// LS Electric XG5000 project: project
// PLC LSPLC

PROGRAM NewProgram (task: 스캔 프로그램)

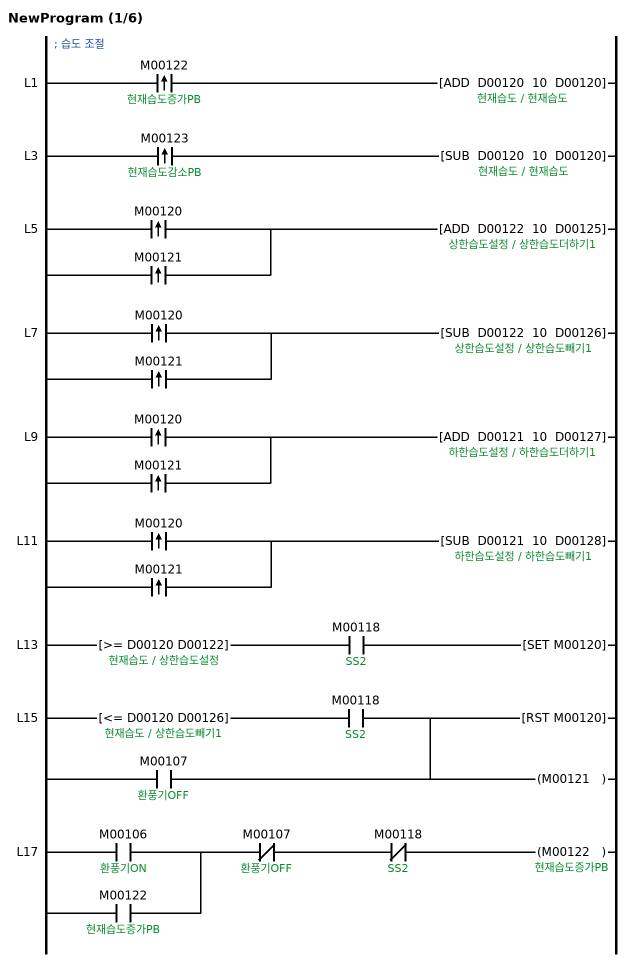
// 습도 조절
; L1
LOADP     M00122	// 현재습도증가PB
ADD       D00120 10 D00120	// 현재습도 / 현재습도
; L3
LOADP     M00123	// 현재습도감소PB
SUB       D00120 10 D00120	// 현재습도 / 현재습도
; L5
LOADP     M00120
ORP       M00121
ADD       D00122 10 D00125	// 상한습도설정 / 상한습도더하기1
; L7
LOADP     M00120
ORP       M00121
SUB       D00122 10 D00126	// 상한습도설정 / 상한습도빼기1
; L9
LOADP     M00120
ORP       M00121
ADD       D00121 10 D00127	// 하한습도설정 / 하한습도더하기1
; L11
LOADP     M00120
ORP       M00121
SUB       D00121 10 D00128	// 하한습도설정 / 하한습도빼기1
; L13
LOAD>=    D00120 D00122	// 현재습도 / 상한습도설정
AND       M00118	// SS2
SET       M00120
; L15
LOAD<=    D00120 D00126	// 현재습도 / 상한습도빼기1
AND       M00118	// SS2
OR        M00107	// 환풍기OFF
RST       M00120
OUT       M00121
; L17
LOAD      M00106	// 환풍기ON
OR        M00122	// 현재습도증가PB
AND NOT   M00107	// 환풍기OFF
AND NOT   M00118	// SS2
OUT       M00122	// 현재습도증가PB

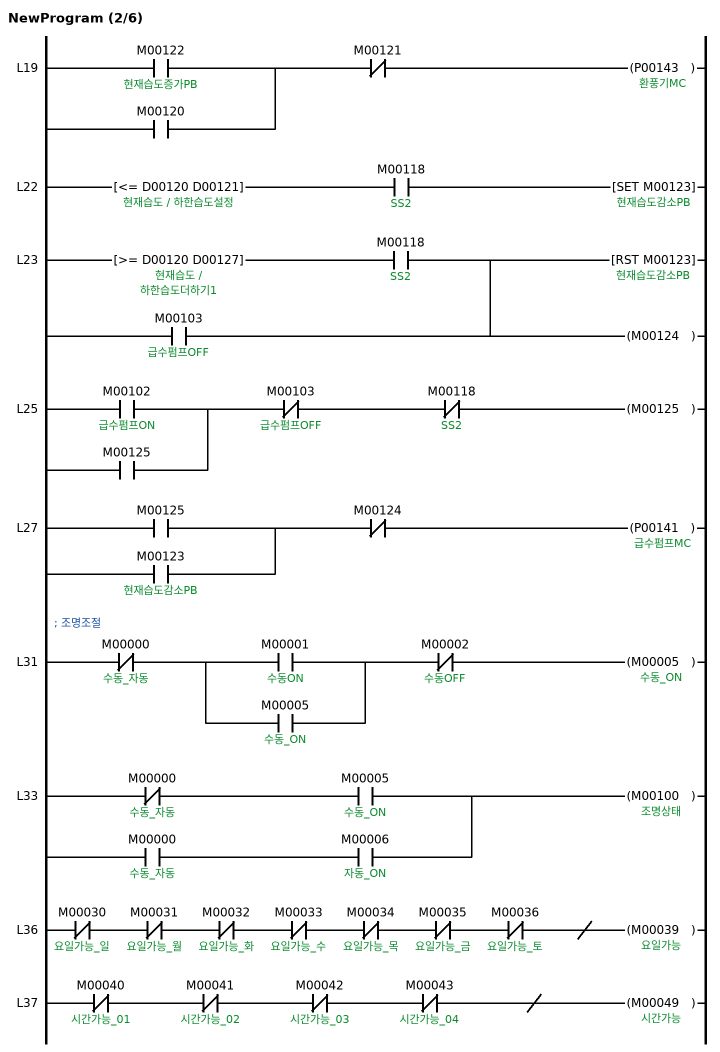
; L19
LOAD      M00122	// 현재습도증가PB
OR        M00120
AND NOT   M00121
OUT       P00143	// 환풍기MC
; L22
LOAD<=    D00120 D00121	// 현재습도 / 하한습도설정
AND       M00118	// SS2
SET       M00123	// 현재습도감소PB
; L23
LOAD>=    D00120 D00127	// 현재습도 / 하한습도더하기1
AND       M00118	// SS2
OR        M00103	// 급수펌프OFF
RST       M00123	// 현재습도감소PB
OUT       M00124
; L25
LOAD      M00102	// 급수펌프ON
OR        M00125
AND NOT   M00103	// 급수펌프OFF
AND NOT   M00118	// SS2
OUT       M00125
; L27
LOAD      M00125
OR        M00123	// 현재습도감소PB
AND NOT   M00124
OUT       P00141	// 급수펌프MC
// 조명조절
; L31
LOAD NOT  M00000	// 수동_자동
LOAD      M00001	// 수동ON
OR        M00005	// 수동_ON
AND LOAD
AND NOT   M00002	// 수동OFF
OUT       M00005	// 수동_ON
; L33
LOAD NOT  M00000	// 수동_자동
AND       M00005	// 수동_ON
LOAD      M00000	// 수동_자동
AND       M00006	// 자동_ON
OR LOAD
OUT       M00100	// 조명상태
; L36
LOAD NOT  M00030	// 요일가능_일
AND NOT   M00031	// 요일가능_월
AND NOT   M00032	// 요일가능_화
AND NOT   M00033	// 요일가능_수
AND NOT   M00034	// 요일가능_목
AND NOT   M00035	// 요일가능_금
AND NOT   M00036	// 요일가능_토
NOT
OUT       M00039	// 요일가능
; L37
LOAD NOT  M00040	// 시간가능_01
AND NOT   M00041	// 시간가능_02
AND NOT   M00042	// 시간가능_03
AND NOT   M00043	// 시간가능_04
NOT
OUT       M00049	// 시간가능

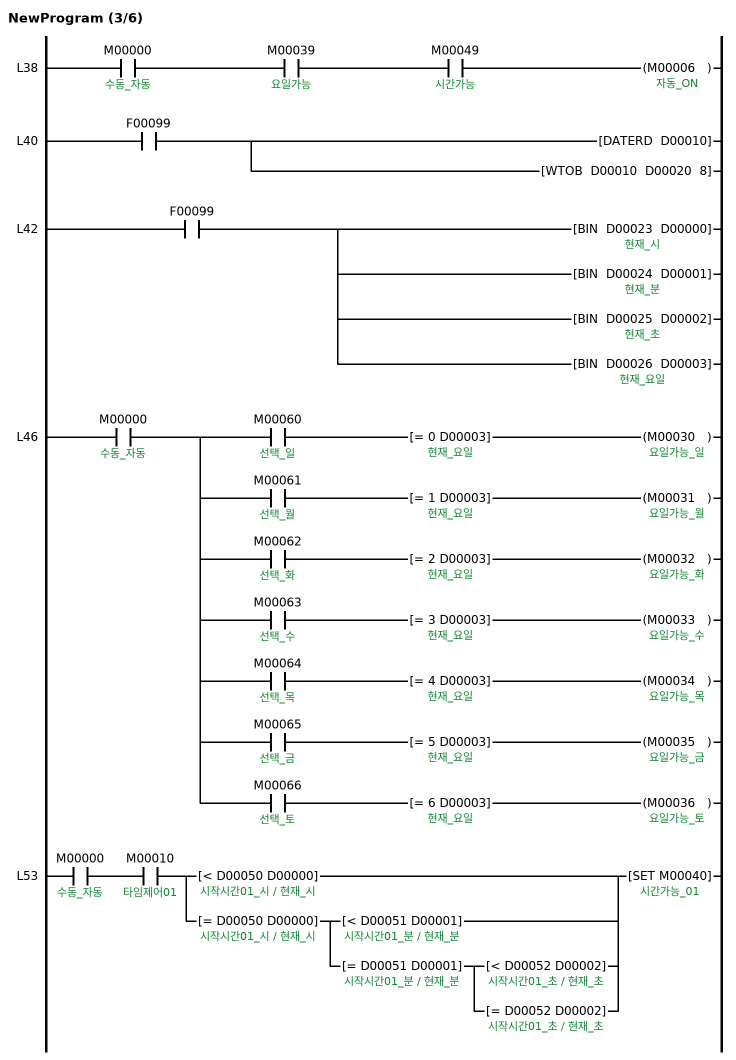
; L38
LOAD      M00000	// 수동_자동
AND       M00039	// 요일가능
AND       M00049	// 시간가능
OUT       M00006	// 자동_ON
; L40
LOAD      F00099
DATERD    D00010
WTOB      D00010 D00020 8
; L42
LOAD      F00099
BIN       D00023 D00000	// 현재_시
BIN       D00024 D00001	// 현재_분
BIN       D00025 D00002	// 현재_초
BIN       D00026 D00003	// 현재_요일
; L46
LOAD      M00000	// 수동_자동
MPUSH
AND       M00060	// 선택_일
AND=      0 D00003	// 현재_요일
OUT       M00030	// 요일가능_일
MLOAD
AND       M00061	// 선택_월
AND=      1 D00003	// 현재_요일
OUT       M00031	// 요일가능_월
MLOAD
AND       M00062	// 선택_화
AND=      2 D00003	// 현재_요일
OUT       M00032	// 요일가능_화
MLOAD
AND       M00063	// 선택_수
AND=      3 D00003	// 현재_요일
OUT       M00033	// 요일가능_수
MLOAD
AND       M00064	// 선택_목
AND=      4 D00003	// 현재_요일
OUT       M00034	// 요일가능_목
MLOAD
AND       M00065	// 선택_금
AND=      5 D00003	// 현재_요일
OUT       M00035	// 요일가능_금
MPOP
AND       M00066	// 선택_토
AND=      6 D00003	// 현재_요일
OUT       M00036	// 요일가능_토
; L53
LOAD      M00000	// 수동_자동
AND       M00010	// 타임제어01
LOAD<     D00050 D00000	// 시작시간01_시 / 현재_시
LOAD=     D00050 D00000	// 시작시간01_시 / 현재_시
LOAD<     D00051 D00001	// 시작시간01_분 / 현재_분
LOAD=     D00051 D00001	// 시작시간01_분 / 현재_분
LOAD<     D00052 D00002	// 시작시간01_초 / 현재_초
OR=       D00052 D00002	// 시작시간01_초 / 현재_초
AND LOAD
OR LOAD
AND LOAD
OR LOAD
AND LOAD
SET       M00040	// 시간가능_01

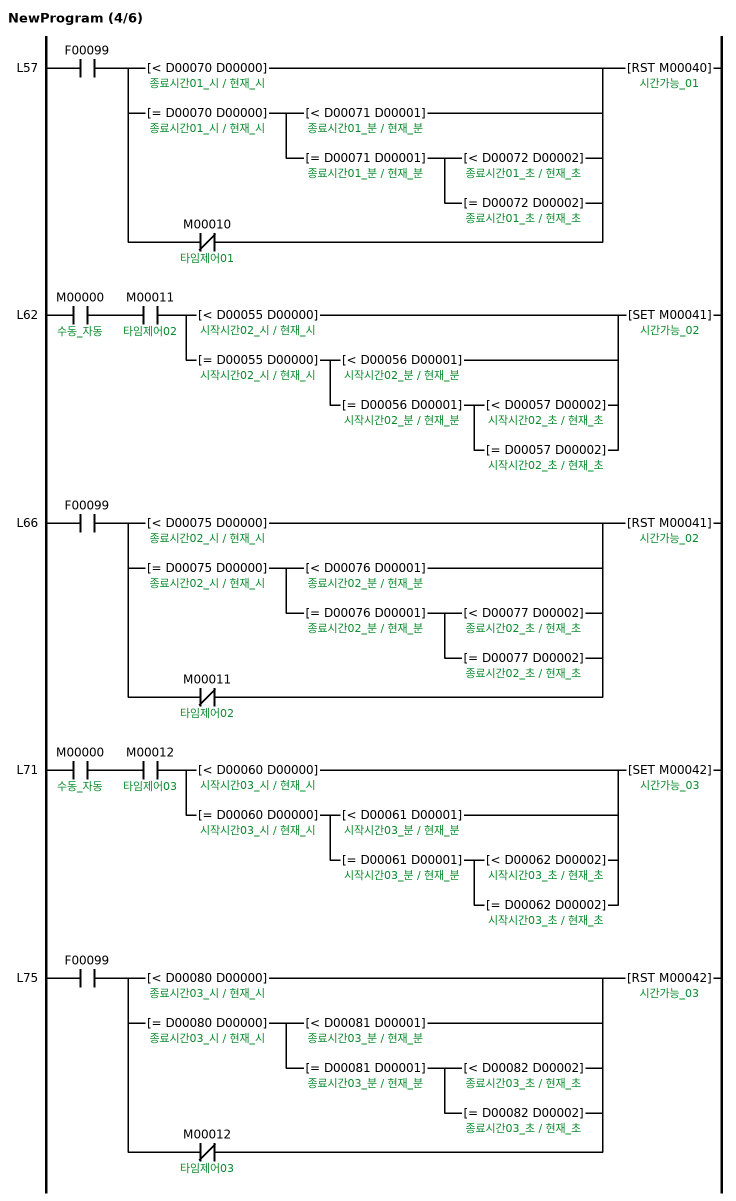
; L57
LOAD      F00099
LOAD<     D00070 D00000	// 종료시간01_시 / 현재_시
LOAD=     D00070 D00000	// 종료시간01_시 / 현재_시
LOAD<     D00071 D00001	// 종료시간01_분 / 현재_분
LOAD=     D00071 D00001	// 종료시간01_분 / 현재_분
LOAD<     D00072 D00002	// 종료시간01_초 / 현재_초
OR=       D00072 D00002	// 종료시간01_초 / 현재_초
AND LOAD
OR LOAD
AND LOAD
OR LOAD
OR NOT    M00010	// 타임제어01
AND LOAD
RST       M00040	// 시간가능_01
; L62
LOAD      M00000	// 수동_자동
AND       M00011	// 타임제어02
LOAD<     D00055 D00000	// 시작시간02_시 / 현재_시
LOAD=     D00055 D00000	// 시작시간02_시 / 현재_시
LOAD<     D00056 D00001	// 시작시간02_분 / 현재_분
LOAD=     D00056 D00001	// 시작시간02_분 / 현재_분
LOAD<     D00057 D00002	// 시작시간02_초 / 현재_초
OR=       D00057 D00002	// 시작시간02_초 / 현재_초
AND LOAD
OR LOAD
AND LOAD
OR LOAD
AND LOAD
SET       M00041	// 시간가능_02
; L66
LOAD      F00099
LOAD<     D00075 D00000	// 종료시간02_시 / 현재_시
LOAD=     D00075 D00000	// 종료시간02_시 / 현재_시
LOAD<     D00076 D00001	// 종료시간02_분 / 현재_분
LOAD=     D00076 D00001	// 종료시간02_분 / 현재_분
LOAD<     D00077 D00002	// 종료시간02_초 / 현재_초
OR=       D00077 D00002	// 종료시간02_초 / 현재_초
AND LOAD
OR LOAD
AND LOAD
OR LOAD
OR NOT    M00011	// 타임제어02
AND LOAD
RST       M00041	// 시간가능_02
; L71
LOAD      M00000	// 수동_자동
AND       M00012	// 타임제어03
LOAD<     D00060 D00000	// 시작시간03_시 / 현재_시
LOAD=     D00060 D00000	// 시작시간03_시 / 현재_시
LOAD<     D00061 D00001	// 시작시간03_분 / 현재_분
LOAD=     D00061 D00001	// 시작시간03_분 / 현재_분
LOAD<     D00062 D00002	// 시작시간03_초 / 현재_초
OR=       D00062 D00002	// 시작시간03_초 / 현재_초
AND LOAD
OR LOAD
AND LOAD
OR LOAD
AND LOAD
SET       M00042	// 시간가능_03
; L75
LOAD      F00099
LOAD<     D00080 D00000	// 종료시간03_시 / 현재_시
LOAD=     D00080 D00000	// 종료시간03_시 / 현재_시
LOAD<     D00081 D00001	// 종료시간03_분 / 현재_분
LOAD=     D00081 D00001	// 종료시간03_분 / 현재_분
LOAD<     D00082 D00002	// 종료시간03_초 / 현재_초
OR=       D00082 D00002	// 종료시간03_초 / 현재_초
AND LOAD
OR LOAD
AND LOAD
OR LOAD
OR NOT    M00012	// 타임제어03
AND LOAD
RST       M00042	// 시간가능_03

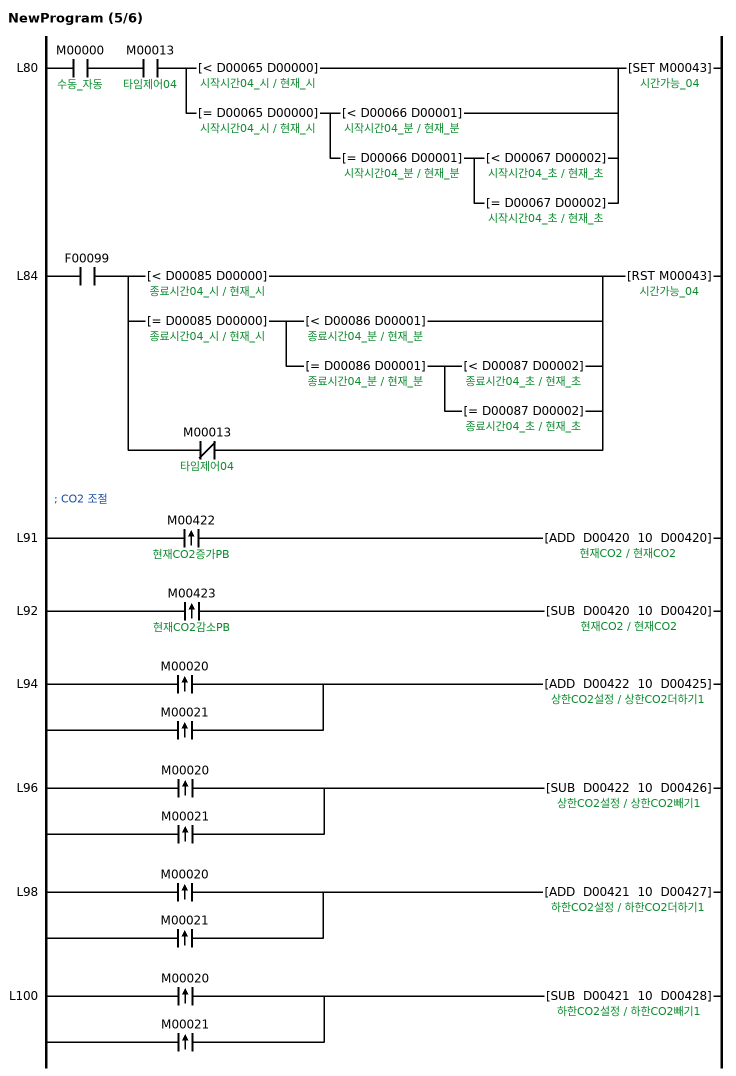
; L80
LOAD      M00000	// 수동_자동
AND       M00013	// 타임제어04
LOAD<     D00065 D00000	// 시작시간04_시 / 현재_시
LOAD=     D00065 D00000	// 시작시간04_시 / 현재_시
LOAD<     D00066 D00001	// 시작시간04_분 / 현재_분
LOAD=     D00066 D00001	// 시작시간04_분 / 현재_분
LOAD<     D00067 D00002	// 시작시간04_초 / 현재_초
OR=       D00067 D00002	// 시작시간04_초 / 현재_초
AND LOAD
OR LOAD
AND LOAD
OR LOAD
AND LOAD
SET       M00043	// 시간가능_04
; L84
LOAD      F00099
LOAD<     D00085 D00000	// 종료시간04_시 / 현재_시
LOAD=     D00085 D00000	// 종료시간04_시 / 현재_시
LOAD<     D00086 D00001	// 종료시간04_분 / 현재_분
LOAD=     D00086 D00001	// 종료시간04_분 / 현재_분
LOAD<     D00087 D00002	// 종료시간04_초 / 현재_초
OR=       D00087 D00002	// 종료시간04_초 / 현재_초
AND LOAD
OR LOAD
AND LOAD
OR LOAD
OR NOT    M00013	// 타임제어04
AND LOAD
RST       M00043	// 시간가능_04
// CO2 조절
; L91
LOADP     M00422	// 현재CO2증가PB
ADD       D00420 10 D00420	// 현재CO2 / 현재CO2
; L92
LOADP     M00423	// 현재CO2감소PB
SUB       D00420 10 D00420	// 현재CO2 / 현재CO2
; L94
LOADP     M00020
ORP       M00021
ADD       D00422 10 D00425	// 상한CO2설정 / 상한CO2더하기1
; L96
LOADP     M00020
ORP       M00021
SUB       D00422 10 D00426	// 상한CO2설정 / 상한CO2빼기1
; L98
LOADP     M00020
ORP       M00021
ADD       D00421 10 D00427	// 하한CO2설정 / 하한CO2더하기1
; L100
LOADP     M00020
ORP       M00021
SUB       D00421 10 D00428	// 하한CO2설정 / 하한CO2빼기1

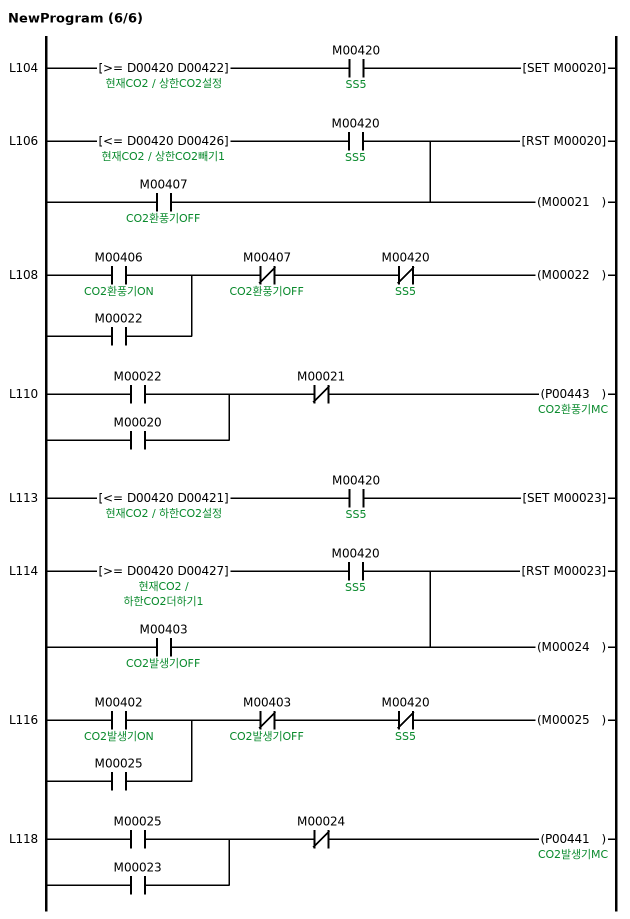
; L104
LOAD>=    D00420 D00422	// 현재CO2 / 상한CO2설정
AND       M00420	// SS5
SET       M00020
; L106
LOAD<=    D00420 D00426	// 현재CO2 / 상한CO2빼기1
AND       M00420	// SS5
OR        M00407	// CO2환풍기OFF
RST       M00020
OUT       M00021
; L108
LOAD      M00406	// CO2환풍기ON
OR        M00022
AND NOT   M00407	// CO2환풍기OFF
AND NOT   M00420	// SS5
OUT       M00022
; L110
LOAD      M00022
OR        M00020
AND NOT   M00021
OUT       P00443	// CO2환풍기MC
; L113
LOAD<=    D00420 D00421	// 현재CO2 / 하한CO2설정
AND       M00420	// SS5
SET       M00023
; L114
LOAD>=    D00420 D00427	// 현재CO2 / 하한CO2더하기1
AND       M00420	// SS5
OR        M00403	// CO2발생기OFF
RST       M00023
OUT       M00024
; L116
LOAD      M00402	// CO2발생기ON
OR        M00025
AND NOT   M00403	// CO2발생기OFF
AND NOT   M00420	// SS5
OUT       M00025
; L118
LOAD      M00025
OR        M00023
AND NOT   M00024
OUT       P00441	// CO2발생기MC